(* CoDeSys 2.3.9.31 project: Test2.pro *)
(* Libraries: STANDARD.LIB 5.6.98 11:03:02 *)

(* Task configuration *)
TASK Standard (PRIORITY := 0, INTERVAL := T#10ms);
	MAIN
END_TASK

(* Global variable list: Global_Variables *)
VAR_GLOBAL
(**DB Address**)
	DB8 AT %MW2010:ARRAY[0..100] OF INT;
(*******用到的数组值有以下变量*******)
(*
	DB8[0],DB8[2],DB8[4],DB8[6],DB8[8],DB8[10],DB8[26],DB8[36],DB8[38],DB8[40],DB8[46],DB8[50],DB8[52],DB8[54],DB8[56],DB8[58],DB8[60],DB8[62],DB8[64],DB8[66],DB8[68],
DB8[70],DB8[72],DB8[74],DB8[76],DB8[78],DB8[80],DB8[82],DB8[84],DB8[86],DB8[88],DB8[90],DB8[92],
*)
(***  MW  Address Define***)
(*	HorizontalManSpeed AT %MW254:INT:=111;
	Man_spd AT %MW260:INT:=222;
	StorageLevel2 AT %MW266:INT:=333;
         GearRatio11 AT %MW270:INT:=411;
         GearRatio22 AT %MW272:INT:=511;
	GearRatio12 AT %MW274:INT:=611;
(***MW1200、MW1202、MW1206、MW1208 ： word(Original)**)
	Pasim_SPEED AT %MW1200:INT:=711;
	PasimFiltSpeed AT %MW1202:INT:=811;
	Packing_SPEED AT %MW1206:INT:=911;
	PackingFiltSpeed AT %MW1208:INT:=121;

        Parsim_speed AT %MW1300:INT:=131;
	MW1302 AT %MW1302: INT:=141;
	MW1304 AT %MW1304:INT:=151;
	MW1310 AT %MW1310:INT:=161;
	MW1250 AT %MW1250:INT:=171;

	MW1534 AT %MW1534:INT:=181;
	MW1536 AT %MW1536:INT:=191;
	MW1634 AT %MW1634:INT:=112;
	MW1636 AT %MW1636:INT:=113;
	MW1734 AT %MW1734:INT:=114;
	MW1736 AT %MW1736:INT:=115;
	MW1738 AT %MW1738:INT:=116;
	MW1740 AT %MW1740:INT:=117;

	MW180 AT %MW180:INT:=118;
	MW182 AT %MW182:INT:=119;
	MW1880 AT %MW1880:INT:=1110;
	MW1884 AT %MW1884:INT:=1111;
	MW1886 AT %MW1886:INT:=1112;

	MW1950 AT %MW1950:INT:=1113;
	MW1952 AT %MW1952:INT:=1114;


	MakerExportActSpeed AT %MW2236:INT:=1115;
     LiftActSpeed AT %MW1936:INT:=1116;
          TransferActSpeed AT %MW2036:INT:=1117;
	MakerExportCigSpeed AT %MW1404:INT:=1118;
          LiftCigSpeed AT %MW1400:INT:=1119;
          TransferCigSpeed AT %MW1402:INT:=555;


	MakerExportFaultNum AT %MW2800:DWORD:=7340;
	SampleFaultNum AT %MW2802:DWORD:=16#733F;
	CornerFaultNum AT %MW2804:DWORD:=5260;
	LiftFaultNum AT %MW2806:DWORD:=5320;
	TransferFaultNum AT %MW2808:DWORD:=6430;
	SlopeFaultNum AT %MW2810:DWORD:=3210;
	StorageFaultNum AT %MW2812:DWORD:=4350;

 (***  MX  Address Define***)
	SampleEntrJammedDis AT %MX50.0:BOOL;
	ElevatorEntrJammedDis AT %MX50.1:BOOL;
	Drop_JammedDis AT %MX50.2:BOOL;
	Axis2OverloadDis AT %MX50.3:BOOL;
	StorageOverloadDis AT %MX50.4:BOOL;
	StorageEntrJammedDis AT %MX50.5:BOOL;
	StorageLimitOn AT %MX60.2:BOOL;
	Storage_Full AT %MX71.2:BOOL;

	M80_0 AT %MX80.0: BOOL;
	PackingRun AT %MX80.1:BOOL;
	EncoderNOFeedback AT %MX71.3:BOOL;
	Man_start AT %MX500.1:BOOL;
	ManEmptyON AT %MX501.0:BOOL;
	Tisheng_Auto_start AT %MX502.1:BOOL;
	cunchu_man_str AT %MX550.1:BOOL;
	cunchu_auto_str AT %MX552.1:BOOL;
	pai_kong_on AT %MX553.7:BOOL;

	EncoderZeroON AT %MX1000.0:BOOL;
	TryRunON AT %MX1000.6:BOOL;
	StorageForceRun AT %MX1000.7:BOOL;
	StorageForceRunBlink AT %MX1002.0:BOOL;

	M1502_5 AT %MX1502.5:BOOL;
	Axis1InitOk  AT %MX1502.7:BOOL;
	M1602_5 AT %MX1602.5:BOOL;
	Axis2InitOk  AT %MX1602.7:BOOL;
	Axis3EnableOut  AT %MX1702.5:BOOL;
	Axis3InitOk  AT %MX1702.7:BOOL;
	M1802_5 AT %MX1802.5:BOOL;
	Axis4InitOk  AT %MX1802.7:BOOL;
	Axis2_1EnableOut  AT %MX1902.5:BOOL;
	Axis2_1InitOk  AT %MX1902.7:BOOL;
	Axis2_2EnableOut  AT %MX2002.5:BOOL;
	Axis2_2InitOk  AT %MX2002.7:BOOL;
	MakerExportEnableOut  AT %MX2102.5:BOOL;
	MakerExportInitOk  AT %MX2102.7:BOOL;

	MakerExportEcError AT %MX2600.0:BOOL;
         SamlpeEcError AT %MX2600.1:BOOL;
	CornerEcError AT %MX2600.2:BOOL;
	LiftEcError AT %MX2600.3:BOOL;
	TransferEcError AT %MX2600.4:BOOL;
	SlopeEcError AT %MX2600.5:BOOL;
	StorageEcError AT %MX2600.6:BOOL;

	AllEmpty AT %MX2603.6:BOOL;
	ManEmpty AT %MX2603.7:BOOL;


	Input1EcError AT %MX2601.1:BOOL;
	Input2EcError AT %MX2601.2:BOOL;
	Input3EcError AT %MX2601.3:BOOL;
	Input4EcError AT %MX2601.4:BOOL;
	Input5EcError AT %MX2601.5:BOOL;
	Input6EcError AT %MX2601.6:BOOL;
	Input7EcError AT %MX2601.7:BOOL;
	Output1EcError AT %MX2602.0:BOOL;
	Output2EcError AT %MX2602.1:BOOL;
	Output3EcError AT %MX2602.2:BOOL;
	Output4EcError AT %MX2602.3:BOOL;
	Analog1EcError AT %MX2602.4:BOOL;
	Analog2EcError AT %MX2602.5:BOOL;

	StoreUnitStop AT %MX2603.0:BOOL;
	ElevaterStop AT %MX2603.1:BOOL;
	ManualRun AT %MX2603.2:BOOL;
	AutoRun AT %MX2603.3:BOOL;
	ElevaterManualRun AT %MX2603.4:BOOL;

	EmergercyStop_CR AT %IX0.0:BOOL;
	CigMakingExportPower AT %IX0.1:BOOL;
	SamplePower AT %IX0.2:BOOL;
	CornerPower AT %IX0.3:BOOL;
	LiftPower AT %IX0.4:BOOL;
	TransferPower AT %IX0.5:BOOL;
	SlopePower AT %IX0.6:BOOL;
	StoragePower AT %IX0.7:BOOL;

	I1_0Spare AT %IX1.0:BOOL;
	I1_1Spare AT %IX1.1:BOOL;
	CigMakingExportError AT %IX1.2:BOOL;
	SampleError AT %IX1.3:BOOL;
	CornerError AT %IX1.4:BOOL;
	LiftError AT %IX1.5:BOOL;
	TransferError AT %IX1.6:BOOL;
	SlopeError AT %IX1.7:BOOL;


	StorageError AT %IX2.0:BOOL;
	I2_1Spare AT %IX2.1:BOOL;
	I2_2Spare AT %IX2.2:BOOL;
	Man_AutoExchange_OP1 AT %IX2.3:BOOL;
	Start_OP1 AT %IX2.4:BOOL;
	Reset_OP1 AT %IX2.5:BOOL;
	Stop_OP1 AT %IX2.6:BOOL;
	EmergercyStop_OP1 AT %IX2.7:BOOL;

	I3_0Spare AT %IX3.0:BOOL;
	I3_1Spare AT %IX3.1:BOOL;
	CigMakingExportCigExist  AT %IX3.2:BOOL;
	SampleIEntranceCigExist  AT %IX3.3:BOOL;
	SampleEntranceJammed  AT %IX3.4:BOOL;(*****Spare*******)
	CornerEntranceJammed AT %IX3.5:BOOL;
	CigMakingExportJammed AT %IX3.6:BOOL;
	I3_7Spare AT %IX3.7:BOOL;

	Man_Auto_OP2 AT %IX4.0:BOOL;
	I4_1Spare AT %IX4.1:BOOL;
	Start_OP2 AT %IX4.2:BOOL;
	Reset_OP2 AT %IX4.3:BOOL;
	Stop_OP2 AT %IX4.4:BOOL;
	EmergercyStop_OP2  AT %IX4.5:BOOL;
	I4_6Spare AT %IX4.6:BOOL;
	I4_7Spare AT %IX4.7:BOOL;


	DropJammed AT %IX5.0:BOOL;
	SlopeEmpty AT %IX5.1:BOOL;
         ElevatedCigExist AT %IX5.2:BOOL;
	TransferOverload_PROX AT %IX5.3:BOOL;
         I5_4Spare AT %IX5.4:BOOL;
	I5_5Spare AT %IX5.5:BOOL;
	I5_6Spare AT %IX5.6:BOOL;
	I5_7Spare AT %IX5.7:BOOL;


	StorageFull_PROX AT %IX6.0:BOOL;
	StorageEmpty_PROX AT %IX6.1:BOOL;
	StorageOverload_PROX AT %IX6.2:BOOL;
	StorageEntranceCigExist AT %IX6.3:BOOL;
	StorageEntranceJammed AT %IX6.4:BOOL;
	StorageLimit AT %IX6.5:BOOL;
	StorageRotating  AT %IX6.6:BOOL;
	StorageMotorEnableIN  AT %IX6.7:BOOL;

(**Outside Output Address Define**)
	SampleEnableOUT  AT %QX4.0:BOOL;
	CornerEnableOUT  AT %QX4.1:BOOL;
	LiftEnableOUT  AT %QX4.2:BOOL;
	TransferEnableOUT AT %QX4.3:BOOL;
	SlopeEnableOUT  AT %QX4.4:BOOL;
	StorageEnableOUT AT %QX4.5:BOOL;
	Q4_6Spare AT %QX4.6:BOOL;
	Q4_7Spare AT %QX4.7:BOOL;

	Start_IndicatorOP1 AT %QX5.0:BOOL;
	Reset_IndicatorOP1 AT %QX5.1:BOOL;
	Stop_IndicatorOP1 AT %QX5.2:BOOL;
	StorageReset AT %QX5.3:BOOL;
	CigMakingPermission AT %QX5.4:BOOL;
	SynTracking AT %QX5.5:BOOL;
	A_BModeExchange AT %QX5.6:BOOL;
	CigMakingEmergStop AT %QX5.7:BOOL;

	StorageShakeTest AT %QX8.0:BOOL;
	Q8_1Spare AT %QX8.1:BOOL;
	PackerPermission AT %QX8.2:BOOL;
	PackerLowVelRequest AT %QX8.3:BOOL;(****Spare*****)
	Q8_4Spare AT %QX8.4:BOOL;
	Q8_5Spare AT %QX8.5:BOOL;
	Q8_6Spare  AT %QX8.6:BOOL;
	Start_Indic_OP2 AT %QX8.7:BOOL;

	Reset_Indic_OP2 AT %QX9.0:BOOL;
	Stop_Indic_OP2 AT %QX9.1:BOOL;
	EmergercyStop_IndicOP2 AT %QX9.2:BOOL;
	StorageFull_IndicOP2 AT %QX9.3:BOOL;
	StorageEmpty_IndicOP2 AT %QX9.4:BOOL;
	StorageOverload_IndicOP2 AT %QX9.5:BOOL;
	StorageLimit_IndicOP2 AT %QX9.6:BOOL;
	StorageEntrJammed_IndicOP2 AT %QX9.7:BOOL;

	DropJammed_IndicOP2 AT %QX10.0:BOOL;
	PackerPerm_IndicOP2 AT %QX10.1:BOOL;
	SlopEmpty_IndicOP2 AT %QX10.2:BOOL;
	SampleEntrJam_Indication AT %QX10.3:BOOL;
	ElevatorEntrJam_Indication AT %QX10.4:BOOL;
	TransferOverload_Indication AT %QX10.5:BOOL;
	CigMakingPerm_IndicOP2 AT %QX10.6:BOOL;
	Q10_7Spare AT %QX10.7:BOOL;

(********************************************************************************************)
	Corner_pid_sp:INT;
	Corner_work_limit:INT;
	Corner_work_off_delay:INT;
	Corner_pid_p_gain:INT;
	Corner_p_parameter:INT;
	cig_dim:INT;
	Store_CigIn_Comp_speed1:INT;
	Store_CigIn_Comp_speed2:INT;
	Downport_CigIn_hight2:INT;
	Corner_pid_i_gain:INT;
	Maker_MaxSpeedLimit:INT;
	Packer_MaxSpeedLimit:INT;
	Store_empty_position:INT;
	Store_full_position:INT;
	Packer_LowSpeed_position:INT;
	Packer_enable_position:INT;
	Maker_stop_position:INT;
	Corner_entrance_hight_limit:INT;
	Corner_entrance_low_limt:INT;
	Downport_CigIn_hight1:INT;
	Corner_pid_deadband:INT;
	Downport_CigOut_hight1:INT;
	Downport_CigOut_hight2:INT;
	Store_CigOut_Comp_speed1:INT;
	Store_CigOut_Comp_speed2:INT;
	Downport_Highest_limit:INT;
	Downport_Lowest_limit:INT;
	Downport_CigIn_lowest_hight:INT;
	Store_set_zero:BOOL;
	test_run:BOOL;
	StoreUnit_discharge_button:BOOL;
	Elevater_man_paikong:BOOL;
	test_run_unprotected:BOOL;
	test_maker_speed:INT;
	test_packer_speed:INT;
	Corner_manual_speed:INT;
	Store_manual_speed:INT;
	Lift_p_parameter:INT;
	Transfer_p_parameter:INT;
	MakerExport_p_parameter:INT;
	Emergency_stop:BOOL;
	MakerExit_power:BOOL;
	Sample_power:BOOL;
	Corner_power:BOOL;
	Lift_power:BOOL;
	Transfer_power:BOOL;
	Slope_power:BOOL;
	Store_power:BOOL;
	Spare10:BOOL;
	Spare11:BOOL;
	MakerExit_servo_fault:BOOL;
	Sample_servo_fault:BOOL;
	Corner_servo_fault:BOOL;
	Lift_servo_fault:BOOL;
	Transfer_servo_fault:BOOL;
	Slope_servo_fault:BOOL;
	Store_servo_fault:BOOL;
	Spare21:BOOL;
	Spare22:BOOL;
	Elevater_man_auto_sw:BOOL;
	Elevater_start_pb:BOOL;
	Elevater_reset_pb:BOOL;
	Elevater_stop_pb:BOOL;
	Elevater_e_stop:BOOL;
	Spare30:BOOL;
	Spare31:BOOL;
	MakerExit_sensor:BOOL;
	Sample_entrance_sensor:BOOL;
	Sample_entrance_jam_sensor:BOOL;
	Corner_entrance_jam_sensor:BOOL;
	MakerExit_jam_sensor:BOOL;
	Spare37:BOOL;
	StoreUnit_man_auto_sw:BOOL;
	Spare41:BOOL;
	StoreUnit_start_button:BOOL;
	StoreUnit_reset_button:BOOL;
	StoreUnit_stop_button:BOOL;
	StoreUnit_e_stop_button:BOOL;
	Spare46:BOOL;
	Spare47:BOOL;
	Downport_jam_sensor:BOOL;
	Slope_empty:BOOL;
	Transfer_cig_exist:BOOL;
	Transfer_overload_sensor:BOOL;
	Spare54:BOOL;
	Spare55:BOOL;
	Spare56:BOOL;
	Spare57:BOOL;
	Store_full:BOOL;
	Store_empty:BOOL;
	Store_overload:BOOL;
	Store_entrance_cig_exist:BOOL;
	Store_entrance_jam:BOOL;
	Store_overlimit:BOOL;
	Store_running:BOOL;
	Store_enabled:BOOL;
	sample_servo_enable_Q:BOOL;
	Corner_servo_enable_Q:BOOL;
	Lift_servo_enable_Q:BOOL;
	Transfer_servo_enable_Q:BOOL;
	Slope_servo_enable_Q:BOOL;
	Store_servo_enable_Q:BOOL;
	SpareOutput46:BOOL;
	SpareOutput47:BOOL;
	Elevater_start_Q:BOOL;
	Elevater_reset_Q:BOOL;
	Elevater_stop_Q:BOOL;
	Elevater_FaultReset_Q:BOOL;
	Maker_enable_relay_Q:BOOL;
	SpareOutput55:BOOL;
	SpareOutput56:BOOL;
	Maker_QuickStop_Q:BOOL;
	SpareOutput80:BOOL;
	SpareOutput81:BOOL;
	Packer_enable_relay_Q:BOOL;
	Packer_LowSpeed_request_Q:BOOL;
	SpareOutput84:BOOL;
	SpareOutput85:BOOL;
	SpareOutput86:BOOL;
	StoreUnit_start_Q:BOOL;
	StoreUnit_reset_Q:BOOL;
	StoreUnit_stop_Q:BOOL;
	SpareOutput92:BOOL;
	SpareOutput93:BOOL;
	SpareOutput94:BOOL;
	SpareOutput95:BOOL;
	SpareOutput96:BOOL;
	SpareOutput97:BOOL;
	MakerExit_servo_enable:BOOL;
	MakerExit_servo_initialized:BOOL;
	sample_servo_enable:BOOL;
	sample_servo_initialized:BOOL;
	Corner_servo_enable:BOOL;
	Corner_servo_initialized:BOOL;
	Slope_servo_enable:BOOL;
	Slope_servo_initialized:BOOL;
	Store_servo_enable:BOOL;
	Lift_servo_enable:BOOL;
	Lift_servo_initialized:BOOL;
	Transfer_servo_enable:BOOL;
	Transfer_servo_initialized:BOOL;
	alarm_sample_entrance_jam:BOOL;
	alarm_corner_entrance_jam:BOOL;
	alarm_downport_entrance_jam:BOOL;
	alarm_transfer_overload:BOOL;
	alarm_store_overload:BOOL;
	alarm_store_entrance_jam:BOOL;
	Elevater_manual_discharge:BOOL;
	Elevater_auto_run:BOOL;
	StoreUnit_man_run:BOOL;
	StoreUnit_auto_run:BOOL;
	StoreUnit_discharge_run:BOOL;
	alarm_store_limit_on:BOOL;
	alarm_store_full:BOOL;
	alarm_encoder_fault:BOOL;
	Maker_run:BOOL;
	packer_run:BOOL;
	MakerExit_servo_ethercat_fault:BOOL;
	Sample_servo_ethercat_fault:BOOL;
	Corner_servo_ethercat_fault:BOOL;
	Lift_servo_ethercat_fault:BOOL;
	Transfer_servo_ethercat_fault:BOOL;
	Slope_servo_ethercat_fault:BOOL;
	Store_servo_ethercat_fault:BOOL;
	Spare26007:BOOL;
	Spare26010:BOOL;
	Digital_Input1_ethercat_fault:BOOL;
	Digital_Input2_ethercat_fault:BOOL;
	Digital_Input3_ethercat_fault:BOOL;
	Digital_Input4_ethercat_fault:BOOL;
	Digital_Input5_ethercat_fault:BOOL;
	Digital_Input6_ethercat_fault:BOOL;
	Digital_Input7_ethercat_fault:BOOL;
	Digital_Output1_ethercat_fault:BOOL;
	Digital_Output2_ethercat_fault:BOOL;
	Digital_Output3_ethercat_fault:BOOL;
	Digital_Output4_ethercat_fault:BOOL;
	Analog_Input1_ethercat_fault:BOOL;
	Analog_Input2_ethercat_fault:BOOL;
	StoreUnit_Stop:BOOL;
	Elevater_Stop:BOOL;
	Manual_Run:BOOL;
	Auto_Run:BOOL;
	Elevater_Manual_Run:BOOL;
	test_run_light:BOOL;
	Corner_pid_output:INT;
	Corner_pid_pv:INT;
	DownPort_hight:INT;
	Store_percent:INT;
	Downport_comp_output:INT;
	Maker_cig_speed:INT;
	Sample_cig_speed:INT;
	Corner_cig_speed:INT;
	Packer_cig_speed:INT;
	Life_cig_speed:INT;
	Transfer_cig_speed:INT;
	MakerExport_cig_speed:INT;
	MakerExport_speed_rpm:INT;
	Sample_speed_rpm:INT;
	Corner_speed_rpm:INT;
	Slope_speed_rpm:INT;
	Store_speed_rpm:INT;
	Corner_entrance_sensor_output:INT;
	Downport_sensor_output:INT;
	Store_CigNum:INT;
	Store_cig_speed:INT;
	Slope_cig_speed:INT;
	Lift_speed_rpm:INT;
	Transfer_speed_rpm:INT;
	MakerExport_Servo_FaultNum:INT;
	Sample_Servo_FaultNum:INT;
	Corner_Servo_FaultNum:INT;
	Lift_Servo_FaultNum:INT;
	Transfer_Servo_FaultNum:INT;
	Slope_Servo_FaultNum:INT;
	Store_Servo_FaultNum:INT;
	Corner_lowlimit:INT;*)




	Store_set_zero AT %MX1000.0 : BOOL;
	test_run AT %MX1000.6 : BOOL;
	StoreUnit_discharge_button AT %MX2603.6 : BOOL;
	Elevater_man_paikong AT %MX2603.7 :BOOL;
	test_run_unprotected AT %MX1000.7 : BOOL;
	test_maker_speed AT %MW1950 : INT;
	test_packer_speed AT %MW1952 : INT;
	Corner_manual_speed AT %MW254 : INT;
	Store_manual_speed AT %MW260 : INT;
	Lift_p_parameter AT %MW270 : INT;
	Transfer_p_parameter AT %MW272 : INT;
	MakerExport_p_parameter AT %MW274 : INT;
	Emergency_stop AT %IX0.0 : BOOL;
	MakerExit_power AT %IX0.1 : BOOL;
	Sample_power AT %IX0.2 : BOOL;
	Corner_power AT %IX0.3 : BOOL;
	Lift_power AT %IX0.4 : BOOL;
	Transfer_power AT %IX0.5 : BOOL;
	Slope_power AT %IX0.6 : BOOL;
	Store_power AT %IX0.7 : BOOL;
	Spare10 AT %IX1.0 : BOOL;
	Spare11 AT %IX1.1 : BOOL;
	MakerExit_servo_fault AT %IX1.2 : BOOL;
	Sample_servo_fault AT %IX1.3 : BOOL;
	Corner_servo_fault AT %IX1.4 : BOOL;
	Lift_servo_fault AT %IX1.5 : BOOL;
	Transfer_servo_fault AT %IX1.6 : BOOL;
	Slope_servo_fault AT %IX1.7 : BOOL;
	Store_servo_fault AT %IX2.0 : BOOL;
	Spare21 AT %IX2.1 : BOOL;
	Spare22 AT %IX2.2 : BOOL;
	Elevater_man_auto_sw AT %IX2.3 : BOOL;
	Elevater_start_pb AT %IX2.4 : BOOL;
	Elevater_reset_pb AT %IX2.5 : BOOL;
	Elevater_stop_pb AT %IX2.6 : BOOL;
	Elevater_e_stop AT %IX2.7 : BOOL;
	Spare30 AT %IX3.0 : BOOL;
	Spare31 AT %IX3.1 : BOOL;
	MakerExit_sensor AT %IX3.2 : BOOL;
	Sample_entrance_sensor AT %IX3.3 : BOOL;
	Sample_entrance_jam_sensor AT %IX3.4 : BOOL;
	Corner_entrance_jam_sensor AT %IX3.5 : BOOL;
	MakerExit_jam_sensor AT %IX3.6 : BOOL;
	Spare37 AT %IX3.7 : BOOL;
	StoreUnit_man_auto_sw AT %IX4.0 : BOOL;
	Spare41 AT %IX4.1 : BOOL;
	StoreUnit_start_button AT %IX4.2 : BOOL;
	StoreUnit_reset_button AT %IX4.3 : BOOL;
	StoreUnit_stop_button AT %IX4.4 : BOOL;
	StoreUnit_e_stop_button AT %IX4.5 : BOOL;
	Spare46 AT %IX4.6 : BOOL;
	Spare47 AT %IX4.7 : BOOL;
	Downport_jam_sensor AT %IX5.0 : BOOL;
	Slope_empty AT %IX5.1 : BOOL;
	Transfer_cig_exist AT %IX5.2 : BOOL;
	Transfer_overload_sensor AT %IX5.3 : BOOL;
	Spare54 AT %IX5.4 : BOOL;
	Spare55 AT %IX5.5 : BOOL;
	Spare56 AT %IX5.6 : BOOL;
	Spare57 AT %IX5.7 : BOOL;
	Store_full AT %IX6.0 : BOOL;
	Store_empty AT %IX6.1 : BOOL;
	Store_overload AT %IX6.2 : BOOL;
	Store_entrance_cig_exist AT %IX6.3 : BOOL;
	Store_entrance_jam AT %IX6.4 : BOOL;
	Store_overlimit AT %IX6.5 : BOOL;
	Store_running AT %IX6.6 : BOOL;
	Store_enabled AT %IX6.7 : BOOL;
	sample_servo_enable_Q AT %QX4.0 : BOOL;
	Corner_servo_enable_Q AT %QX4.1 : BOOL;
	Lift_servo_enable_Q AT %QX4.2 : BOOL;
	Transfer_servo_enable_Q AT %QX4.3 : BOOL;
	Slope_servo_enable_Q AT %QX4.4 : BOOL;
	Store_servo_enable_Q AT %QX4.5 : BOOL;
	SpareOutput46 AT %QX4.6 : BOOL;
	SpareOutput47 AT %QX4.7 : BOOL;
	Elevater_start_Q AT %QX5.0 : BOOL;
	Elevater_reset_Q AT %QX5.1 : BOOL;
	Elevater_stop_Q AT %QX5.2 : BOOL;
	Elevater_FaultReset_Q AT %QX5.3 : BOOL;
	Maker_enable_relay_Q AT %QX5.4 : BOOL;
	SpareOutput55 AT %QX5.5 : BOOL;
	SpareOutput56 AT %QX5.6 : BOOL;
	Maker_QuickStop_Q AT %QX5.7 : BOOL;
	SpareOutput80 AT %QX8.0 : BOOL;
	SpareOutput81 AT %QX8.1 : BOOL;
	Packer_enable_relay_Q AT %QX8.2 : BOOL;
	Packer_LowSpeed_request_Q AT %QX8.3 : BOOL;
	SpareOutput84 AT %QX8.4 : BOOL;
	SpareOutput85 AT %QX8.5 : BOOL;
	SpareOutput86 AT %QX8.6 : BOOL;
	StoreUnit_start_Q AT %QX8.7 : BOOL;
	StoreUnit_reset_Q AT %QX9.0 : BOOL;
	StoreUnit_stop_Q AT %QX9.1 : BOOL;
	SpareOutput92 AT %QX9.2 : BOOL;
	SpareOutput93 AT %QX9.3 : BOOL;
	SpareOutput94 AT %QX9.4 : BOOL;
	SpareOutput95 AT %QX9.5 : BOOL;
	SpareOutput96 AT %QX9.6 : BOOL;
	SpareOutput97 AT %QX9.7 : BOOL;
	MakerExit_servo_enable AT %MX2102.5 : BOOL;
	MakerExit_servo_initialized AT %MX2102.7 : BOOL;
	sample_servo_enable AT %MX1502.5 : BOOL;
	sample_servo_initialized AT %MX1502.7 : BOOL;
	Corner_servo_enable AT %MX1602.5 : BOOL;
	Corner_servo_initialized AT %MX1602.7 : BOOL;
	Slope_servo_enable AT %MX1702.5 : BOOL;
	Slope_servo_initialized AT %MX1702.7 : BOOL;
	Store_servo_enable AT %MX1802.5 : BOOL;
	Lift_servo_enable AT %MX1902.5 : BOOL;
	Lift_servo_initialized AT %MX1902.7 : BOOL;
	Transfer_servo_enable AT %MX2002.5 : BOOL;
	Transfer_servo_initialized AT %MX2002.7 : BOOL;
	alarm_sample_entrance_jam AT %MX50.0 : BOOL;
	alarm_corner_entrance_jam AT %MX50.1 : BOOL;
	alarm_downport_entrance_jam AT %MX50.2 : BOOL;
	alarm_transfer_overload AT %MX50.3 : BOOL;
	alarm_store_overload AT %MX50.4 : BOOL;
	alarm_store_entrance_jam AT %MX50.5 : BOOL;
	Elevater_manual_discharge AT %MX501.0 : BOOL;
	Elevater_auto_run AT %MX502.1 : BOOL;
	StoreUnit_man_run AT %MX550.1 : BOOL;
	StoreUnit_auto_run AT %MX552.1 : BOOL;
	StoreUnit_discharge_run AT %MX553.7 : BOOL;
	alarm_store_limit_on AT %MX60.2 : BOOL;
	alarm_store_full AT %MX71.2 : BOOL;
	alarm_encoder_fault AT %MX71.3 : BOOL;
	Maker_run AT %MX80.0 : BOOL;
	packer_run AT %MX80.1 : BOOL;
	MakerExit_servo_ethercat_fault AT %MX2600.0 : BOOL;
	Sample_servo_ethercat_fault AT %MX2600.1 : BOOL;
	Corner_servo_ethercat_fault AT %MX2600.2 : BOOL;
	Lift_servo_ethercat_fault AT %MX2600.3 : BOOL;
	Transfer_servo_ethercat_fault AT %MX2600.4 : BOOL;
	Slope_servo_ethercat_fault AT %MX2600.5 : BOOL;
	Store_servo_ethercat_fault AT %MX2600.6 : BOOL;
	Spare26007 AT %MX2600.7 : BOOL;
	Spare26010 AT %MX2601.0 : BOOL;
	Digital_Input1_ethercat_fault AT %MX2601.1 : BOOL;
	Digital_Input2_ethercat_fault AT %MX2601.2 : BOOL;
	Digital_Input3_ethercat_fault AT %MX2601.3 : BOOL;
	Digital_Input4_ethercat_fault AT %MX2601.4 : BOOL;
	Digital_Input5_ethercat_fault AT %MX2601.5 : BOOL;
	Digital_Input6_ethercat_fault AT %MX2601.6 : BOOL;
	Digital_Input7_ethercat_fault AT %MX2601.7 : BOOL;
	Digital_Output1_ethercat_fault AT %MX2602.0 : BOOL;
	Digital_Output2_ethercat_fault AT %MX2602.1 : BOOL;
	Digital_Output3_ethercat_fault AT %MX2602.2 : BOOL;
	Digital_Output4_ethercat_fault AT %MX2602.3 : BOOL;
	Analog_Input1_ethercat_fault AT %MX2602.4 : BOOL;
	Analog_Input2_ethercat_fault AT %MX2602.5 : BOOL;
	StoreUnit_Stop AT %MX2603.0 : BOOL;
	Elevater_Stop AT %MX2603.1 : BOOL;
	Manual_Run AT %MX2603.2 : BOOL;
	Auto_Run AT %MX2603.3 : BOOL;
	Elevater_Manual_Run AT %MX2603.4 : BOOL;
	test_run_light AT %MX1002.0 : BOOL;
	Downport_comp_output AT %MW1250 : INT;
	Maker_cig_speed AT %MW1300 : INT;
	Sample_cig_speed AT %MW1302 : INT;
	Corner_cig_speed AT %MW1304 : INT;
	Packer_cig_speed AT %MW1310 : INT;
	Life_cig_speed AT %MW1400 : INT;
	Transfer_cig_speed AT %MW1402 : INT;
	MakerExport_cig_speed AT %MW1404 : INT;
	MakerExport_speed_rpm AT %MW2236 : INT;
	Sample_speed_rpm AT %MW1536 : INT;
	Corner_speed_rpm AT %MW1636 : INT;
	Slope_speed_rpm AT %MW1736 : INT;
	Store_speed_rpm AT %MW1738 : INT;
	Corner_entrance_sensor_output AT %MW180 : INT;
	Downport_sensor_output AT %MW182 : INT;
	Store_CigNum AT %MW1880 : INT;
	Store_cig_speed AT %MW1884 : INT;
	Slope_cig_speed AT %MW1886 : INT;
	Lift_speed_rpm AT %MW1936 : INT;
	Transfer_speed_rpm AT %MW2036 : INT;
	MakerExport_Servo_FaultNum AT %MW2800 : DWORD;
	Sample_Servo_FaultNum AT %MW2802 : DWORD;
	Corner_Servo_FaultNum AT %MW2804 : DWORD;
	Lift_Servo_FaultNum AT %MW2806 : DWORD;

	Transfer_Servo_FaultNum AT %MW2808 : DWORD;
	Slope_Servo_FaultNum AT %MW2810 : DWORD;
	Store_Servo_FaultNum AT %MW2812 : DWORD;





	Corner_pid_sp:INT;
	Corner_work_limit:INT;
	Corner_work_off_delay:INT;
	Corner_pid_p_gain:INT;
	Corner_p_parameter:INT;
	cig_dim:INT;
	Store_CigIn_Comp_speed1:INT;
	Store_CigIn_Comp_speed2:INT;
	Downport_CigIn_hight2:INT;
	Corner_pid_i_gain:INT;
	Maker_MaxSpeedLimit:INT;
	Packer_MaxSpeedLimit:INT;
	Store_empty_position:INT;
	Store_full_position:INT;
	Packer_LowSpeed_position:INT;
	Packer_enable_position:INT;
	Maker_stop_position:INT;
	Corner_entrance_hight_limit:INT;
	Corner_entrance_low_limt:INT;
	Downport_CigIn_hight1:INT;
	Corner_pid_deadband:INT;
	Downport_CigOut_hight1:INT;
	Downport_CigOut_hight2:INT;
	Store_CigOut_Comp_speed1:INT;
	Store_CigOut_Comp_speed2:INT;
	Downport_Highest_limit:INT;
	Downport_Lowest_limit:INT;
	Downport_CigIn_lowest_hight:INT;
	Corner_pid_output:INT;
	Corner_pid_pv:INT;
	DownPort_hight:INT;
	Store_percent:INT;
	Corner_lowlimit:INT;


	WriteFlag:BOOL;

END_VAR

(* POU MAIN, ST *)
PROGRAM MAIN
VAR
	aTON: TON;
	bTON: TON;
	Flag: BOOL := TRUE;
END_VAR
(*aTON(IN:=bTON.Q , PT:=T#200ms , Q=> , ET=> );
bTON(IN:= NOT aTON.Q , PT:=T#200ms , Q=> , ET=> );
Man_Auto_OP2:=bTON.Q;
*)

;

IF WriteFlag THEN

	DB8[0]:=Corner_pid_sp;
	DB8[36]:=Corner_work_limit;
	DB8[38]:=Corner_work_off_delay;
	DB8[4]:=Corner_pid_p_gain;
	DB8[40]:=Corner_p_parameter;
	DB8[46]:=cig_dim;
	DB8[52]:=Store_CigIn_Comp_speed1;
	DB8[54]:=Store_CigIn_Comp_speed2;
	DB8[56]:=Downport_CigIn_hight2;
	DB8[6]:=Corner_pid_i_gain;
	DB8[60]:=Maker_MaxSpeedLimit;
	DB8[62]:=Packer_MaxSpeedLimit;
	DB8[64]:=Store_empty_position;
	DB8[66]:=Store_full_position;
	DB8[68]:=Packer_LowSpeed_position;
	DB8[70]:=Packer_enable_position;
	DB8[72]:=Maker_stop_position;
	DB8[74]:=Corner_entrance_hight_limit;
	DB8[76]:=Corner_entrance_low_limt;
	DB8[78]:=Downport_CigIn_hight1;
	DB8[8]:=Corner_pid_deadband;
	DB8[80]:=Downport_CigOut_hight1;
	DB8[82]:=Downport_CigOut_hight2;
	DB8[84]:=Store_CigOut_Comp_speed1;
	DB8[86]:=Store_CigOut_Comp_speed2;
	DB8[88]:=Downport_Highest_limit;
	DB8[90]:=Downport_Lowest_limit;
	DB8[92]:=Downport_CigIn_lowest_hight;
	
	DB8[10]:=Corner_pid_output;
	DB8[2]:=Corner_pid_pv;
	DB8[26]:=DownPort_hight;
	DB8[50]:=Store_percent;
	
	DB8[58]:=Corner_lowlimit;

	WriteFlag:=0;
ELSE


	Corner_pid_sp:=DB8[0];
	Corner_work_limit:=DB8[36];
	Corner_work_off_delay:=DB8[38];
	Corner_pid_p_gain:=DB8[4];
	Corner_p_parameter:=DB8[40];
	cig_dim:=DB8[46];
	Store_CigIn_Comp_speed1:=DB8[52];
	Store_CigIn_Comp_speed2:=DB8[54];
	Downport_CigIn_hight2:=DB8[56];
	Corner_pid_i_gain:=DB8[6];
	Maker_MaxSpeedLimit:=DB8[60];
	Packer_MaxSpeedLimit:=DB8[62];
	Store_empty_position:=DB8[64];
	Store_full_position:=DB8[66];
	Packer_LowSpeed_position:=DB8[68];
	Packer_enable_position:=DB8[70];
	Maker_stop_position:=DB8[72];
	Corner_entrance_hight_limit:=DB8[74];
	Corner_entrance_low_limt:=DB8[76];
	Downport_CigIn_hight1:=DB8[78];
	Corner_pid_deadband:=DB8[8];
	Downport_CigOut_hight1:=DB8[80];
	Downport_CigOut_hight2:=DB8[82];
	Store_CigOut_Comp_speed1:=DB8[84];
	Store_CigOut_Comp_speed2:=DB8[86];
	Downport_Highest_limit:=DB8[88];
	Downport_Lowest_limit:=DB8[90];
	Downport_CigIn_lowest_hight:=DB8[92];
	
	Corner_pid_output:=DB8[10];
	Corner_pid_pv:=DB8[2];
	DownPort_hight:=DB8[26];
	Store_percent:=DB8[50];
	
	Corner_lowlimit:=DB8[58];

END_IF
END_PROGRAM
